// TIA Portal V20 export
FUNCTION "FIT100_Liter" : Void   // FC27, FBD
{ S7_Optimized_Access := 'TRUE' }
// stored: SetENOAutomatically false
BEGIN

REGION Network 1: Channel input
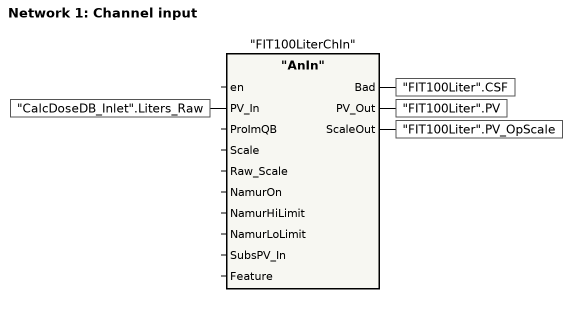
   "FIT100LiterChIn"(PV_In := "CalcDoseDB_Inlet".Liters_Raw,   // "AnIn"
                     Bad => "FIT100Liter".CSF,
                     PV_Out => "FIT100Liter".PV,
                     ScaleOut => "FIT100Liter".PV_OpScale);
END_REGION

REGION Network 2: MonAnL
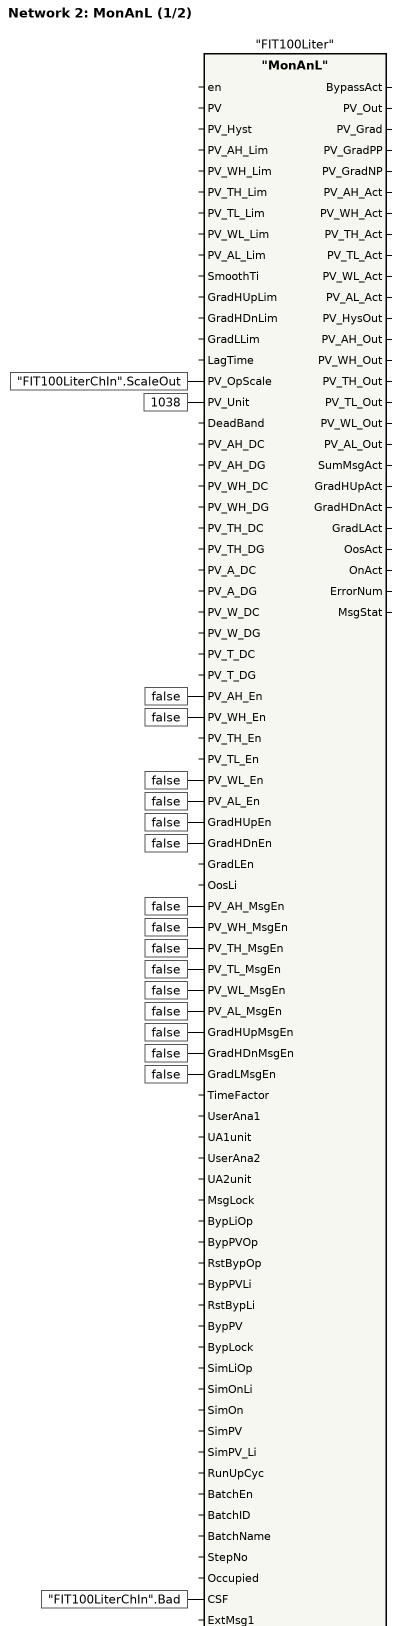
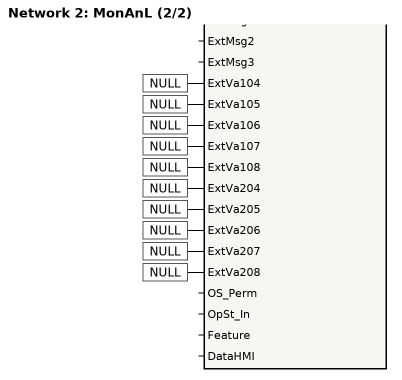
   "FIT100Liter"(PV_OpScale := "FIT100LiterChIn".ScaleOut,   // "MonAnL"
                 PV_Unit := 1038,
                 PV_AH_En := false,
                 PV_WH_En := false,
                 PV_WL_En := false,
                 PV_AL_En := false,
                 GradHUpEn := false,
                 GradHDnEn := false,
                 PV_AH_MsgEn := false,
                 PV_WH_MsgEn := false,
                 PV_TH_MsgEn := false,
                 PV_TL_MsgEn := false,
                 PV_WL_MsgEn := false,
                 PV_AL_MsgEn := false,
                 GradHUpMsgEn := false,
                 GradHDnMsgEn := false,
                 GradLMsgEn := false,
                 CSF := "FIT100LiterChIn".Bad,
                 ExtVa104 := NULL,
                 ExtVa105 := NULL,
                 ExtVa106 := NULL,
                 ExtVa107 := NULL,
                 ExtVa108 := NULL,
                 ExtVa204 := NULL,
                 ExtVa205 := NULL,
                 ExtVa206 := NULL,
                 ExtVa207 := NULL,
                 ExtVa208 := NULL);
END_REGION

REGION Network 3: MTP
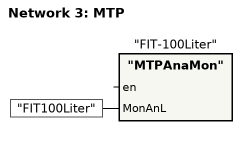
   "FIT-100Liter"(MonAnL := "FIT100Liter");   // "MTPAnaMon"
END_REGION
END_FUNCTION
